{attribute 'qualified_only'}
{attribute 'strict'}
TYPE MOTION_STATUS :
(
	ConstantVelocity := 0,
	Accelerating := 1,
	Decelerating :=2
);
END_TYPE

(* stored: Version 1.1.0.1, ProductVersion 3.1.4024.12
   DUT MOTION_STATUS: Id {f1a60187-137f-40c8-b5c4-a62b7728468b} *)
